// SIMATIC STEP 7 (V5.x) project SterowanieSIlnikiem
// CPU: CPU 317F-2 PN/DP
// station: Hardware
// station: SIMATIC 300
// station: P_ADR_BUS
// program: S7 Program(1)

SYMBOL_TABLE
"CTRL_MOTOR_FWD_BWD"	FC 1	FC 1	// motor control: forward and backward movement
END_SYMBOL_TABLE

FUNCTION "CTRL_MOTOR_FWD_BWD" : VOID	// FC 1
TITLE = sterowanie kierunkiem obrotów silnika elektrycznego
VERSION : 0.1
VAR_INPUT
  Fwd : BOOL ;	//"prawe" obroty silnika: "1" stanem aktywnym
  Bwd : BOOL ;	//"lewe" obroty silnika: "1" stanem aktywnym
  EStop : BOOL ;	//sygna³ z wy³¹cznika awaryjnego: "1" stanem bezpiecznym
  ThermalFuse : BOOL ;	//sygna³ z wy³acznika termicznego: "1" stanem aktywnym
  FwdLSwitch : BOOL ;	//sygna³ z wy³¹cznika krañcowego dla "prawych" obrotów silnika: "1" stanem aktywn
  BwdLSwitch : BOOL ;	//sygna³ z wy³¹cznika krañcowego dla "lewych" obrotów silnika: "1" stanem aktywny
  EStopReset : BOOL ;	//sygna³ resetuj¹cy zadzia³anie wy³¹cznika awaryjnego: zbocze / stanem aktywnym
  ThermalFaultDly : S5TIME ;	//czas wy³¹czenia silnika po zadzia³aniu wy³¹cznika termicznego
  TurnDly : S5TIME ;	//czas wy³¹czenia silnika pomiêdzy kolejnymi rozruchami
  TimerNo1 : TIMER ;	//timer odmierzaj¹cy czas po zadzia³aniu wy³¹cznika termicznego
  TimerNo2 : TIMER ;	//timer odmierzaj¹cy czas pomiêdzy kolejnymi rozruchami
END_VAR
VAR_OUTPUT
  FwdQ : BOOL ;	//"prawe" obroty silnika
  BwdQ : BOOL ;	//"lewe" obroty silnika
  Alarm : BOOL ;	//b³¹d
END_VAR
VAR_IN_OUT
  EStopMem : BOOL ;	//pamiêæ zadzia³ania wy³¹cznika bezpieczeñstwa: "0" stanem bezpiecznym
  EStopResetMem : BOOL ;	//pamiêæ detekcji zbocza na wejœciu EStopReset
  FwdQMem : BOOL ;	//pamiêæ "prawych" obrotów silnika
  BwdQMem : BOOL ;	//pamiêæ "lewych" obrotów silnika
  TurnMem : BOOL ;	//pamiêæ detekcji zbocza wy³¹czenia silnika
END_VAR
VAR_TEMP
  MoveEn : BOOL ;	//zezwolenie na ruch silnika
  ThermalFault : BOOL ;	//zbyt wysoka temperatura silnika
  Turn : BOOL ;	//przerwa do kolejnego rozruchu
END_VAR
BEGIN
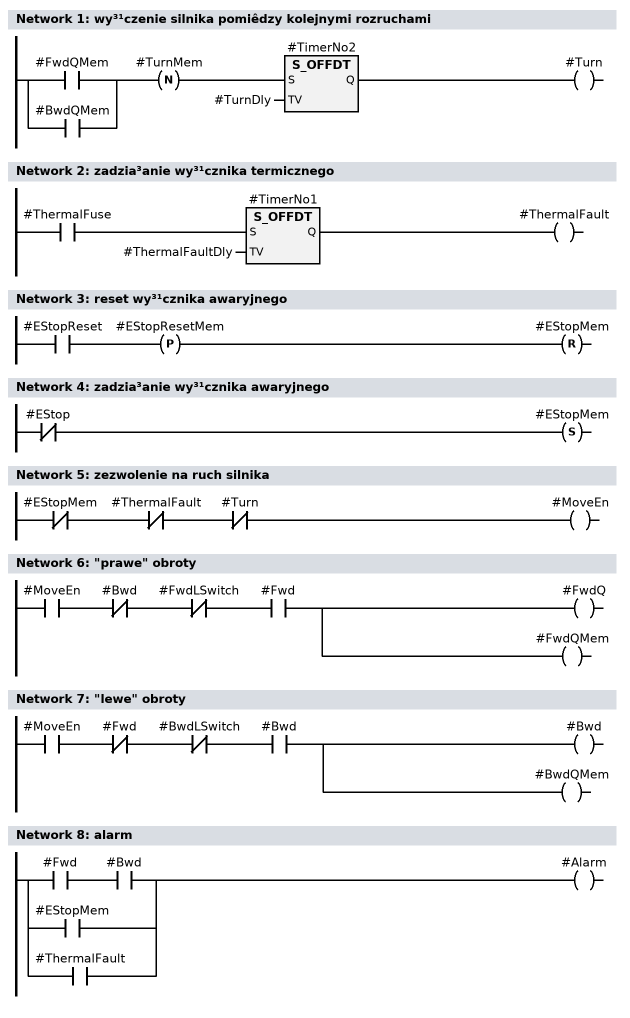
NETWORK
TITLE = wy³¹czenie silnika pomiêdzy kolejnymi rozruchami
//cel:
// - ochrona przed zbyt czêstymi rozruchami silnika
// - czas martwy pomiêdzy zmian¹ kierunku obrotu silnika umo¿liwiaj¹cy 
//prze³¹czenie siê styczników, jak i wyhamowanie silnika
      A(;
      O     #FwdQMem;
      O     #BwdQMem;
      );
      FN    #TurnMem;
      L     #TurnDly;
      SF    #TimerNo2;
      NOP   0;
      NOP   0;
      NOP   0;
      A     #TimerNo2;
      =     #Turn;
NETWORK
TITLE = zadzia³anie wy³¹cznika termicznego
//cel:
// - uniemo¿liwienie za³¹czenia nagrzanego silnika
//
      A     #ThermalFuse;
      L     #ThermalFaultDly;
      SF    #TimerNo1;
      NOP   0;
      NOP   0;
      NOP   0;
      A     #TimerNo1;
      =     #ThermalFault;
NETWORK
TITLE = reset wy³¹cznika awaryjnego
//cel:
// - ochrona przed sta³ym resetowaniem funkcji
// - zmiana logiki dzia³ania na pozytywn¹
      A     #EStopReset;
      FP    #EStopResetMem;
      R     #EStopMem;
NETWORK
TITLE = zadzia³anie wy³¹cznika awaryjnego
// cel:
// - zmiana logiki dzia³ania na pozytywn¹
      AN    #EStop;
      S     #EStopMem;
NETWORK
TITLE = zezwolenie na ruch silnika
//uwaga:
// - nale¿y ustawiæ wartoœæ pocz¹tkow¹ bitu pamiêci EStopMem na "0"
//cel:
// - wypracaowanie pozwolenia na ruch niezwi¹zanego z kierunkiem obrotów silnika
      AN    #EStopMem;
      AN    #ThermalFault;
      AN    #Turn;
      =     #MoveEn;
NETWORK
TITLE = "prawe" obroty
      A     #MoveEn;
      AN    #Bwd;
      AN    #FwdLSwitch;
      A     #Fwd;
      =     #FwdQ;
      =     #FwdQMem;
NETWORK
TITLE = "lewe" obroty
      A     #MoveEn;
      AN    #Fwd;
      AN    #BwdLSwitch;
      A     #Bwd;
      =     #Bwd;
      =     #BwdQMem;
NETWORK
TITLE = alarm
//cel:
// - informacja o jednoczesnym wysterowaniu Fwd i Bwd
// - informacja o wyzwoleniu EStop
// - informacja o zadzia³aniu wy³¹cznika termicznego
      A     #Fwd;
      A     #Bwd;
      O     #EStopMem;
      O     #ThermalFault;
      =     #Alarm;
END_FUNCTION

ORGANIZATION_BLOCK OB 1
TITLE = "Main Program Sweep (Cycle)"
VERSION : 0.1
VAR_TEMP
  OB1_EV_CLASS : BYTE ;	//Bits 0-3 = 1 (Coming event), Bits 4-7 = 1 (Event class 1)
  OB1_SCAN_1 : BYTE ;	//1 (Cold restart scan 1 of OB 1), 3 (Scan 2-n of OB 1)
  OB1_PRIORITY : BYTE ;	//Priority of OB Execution
  OB1_OB_NUMBR : BYTE ;	//1 (Organization block 1, OB1)
  OB1_RESERVED_1 : BYTE ;	//Reserved for system
  OB1_RESERVED_2 : BYTE ;	//Reserved for system
  OB1_PREV_CYCLE : INT ;	//Cycle time of previous OB1 scan (milliseconds)
  OB1_MIN_CYCLE : INT ;	//Minimum cycle time of OB1 (milliseconds)
  OB1_MAX_CYCLE : INT ;	//Maximum cycle time of OB1 (milliseconds)
  OB1_DATE_TIME : DATE_AND_TIME ;	//Date and time OB1 started
END_VAR
BEGIN
// (block stored without names or comments; labels and parameter names are numbered)
END_ORGANIZATION_BLOCK
